FUNCTION_BLOCK FB_ST_HMICommand_Test EXTENDS TcUnit.FB_TestSuite
VAR_INPUT
END_VAR
VAR_OUTPUT
END_VAR
VAR
	testCommand : ST_HMICommand;
END_VAR

// Test runner - call all test methods
Test_InitialState();
Test_EnableCommand();
Test_DisableCommand();
Test_ResetCommand();
Test_StopCommand();
Test_TriggerCommand();
Test_ErrorCode();
Test_MultipleCommands();
Test_ClearCommands();

METHOD Test_ClearCommands
VAR_INPUT
END_VAR
TEST('Test_ClearCommands');

// Set all commands
testCommand.Enable := TRUE;
testCommand.Disable := TRUE;
testCommand.Reset := TRUE;
testCommand.Stop := TRUE;
testCommand.Trigger := TRUE;
testCommand.Error := 42;

// Clear all commands
testCommand.Enable := FALSE;
testCommand.Disable := FALSE;
testCommand.Reset := FALSE;
testCommand.Stop := FALSE;
testCommand.Trigger := FALSE;
testCommand.Error := 0;

// Verify all are cleared
AssertFalse(testCommand.Enable, 'Enable should be FALSE');
AssertFalse(testCommand.Disable, 'Disable should be FALSE');
AssertFalse(testCommand.Reset, 'Reset should be FALSE');
AssertFalse(testCommand.Stop, 'Stop should be FALSE');
AssertFalse(testCommand.Trigger, 'Trigger should be FALSE');
AssertEquals_BYTE(0, testCommand.Error, 'Error should be 0');

TEST_FINISHED();
END_METHOD

METHOD Test_DisableCommand
VAR_INPUT
END_VAR
TEST('Test_DisableCommand');

// Test Disable command can be set
testCommand.Disable := TRUE;
AssertTrue(testCommand.Disable, 'Disable should be TRUE when set');

// Reset
testCommand.Disable := FALSE;
AssertFalse(testCommand.Disable, 'Disable should be FALSE when reset');

TEST_FINISHED();
END_METHOD

METHOD Test_EnableCommand
VAR_INPUT
END_VAR
TEST('Test_EnableCommand');

// Test Enable command can be set
testCommand.Enable := TRUE;
AssertTrue(testCommand.Enable, 'Enable should be TRUE when set');

// Reset
testCommand.Enable := FALSE;
AssertFalse(testCommand.Enable, 'Enable should be FALSE when reset');

TEST_FINISHED();
END_METHOD

METHOD Test_ErrorCode
VAR_INPUT
END_VAR
TEST('Test_ErrorCode');

// Test Error code can be set to various values
testCommand.Error := 0;
AssertEquals_BYTE(0, testCommand.Error, 'Error should be 0');

testCommand.Error := 1;
AssertEquals_BYTE(1, testCommand.Error, 'Error should be 1');

testCommand.Error := 255;
AssertEquals_BYTE(255, testCommand.Error, 'Error should be 255');

testCommand.Error := 128;
AssertEquals_BYTE(128, testCommand.Error, 'Error should be 128');

TEST_FINISHED();
END_METHOD

METHOD Test_InitialState
VAR_INPUT
END_VAR
TEST('Test_InitialState');

// Test that all command flags are initially FALSE
testCommand.Enable := FALSE;
testCommand.Disable := FALSE;
testCommand.Reset := FALSE;
testCommand.Stop := FALSE;
testCommand.Trigger := FALSE;
testCommand.Error := 0;

AssertFalse(testCommand.Enable, 'Enable should be FALSE initially');
AssertFalse(testCommand.Disable, 'Disable should be FALSE initially');
AssertFalse(testCommand.Reset, 'Reset should be FALSE initially');
AssertFalse(testCommand.Stop, 'Stop should be FALSE initially');
AssertFalse(testCommand.Trigger, 'Trigger should be FALSE initially');
AssertEquals_BYTE(0, testCommand.Error, 'Error should be 0 initially');

TEST_FINISHED();
END_METHOD

METHOD Test_MultipleCommands
VAR_INPUT
END_VAR
TEST('Test_MultipleCommands');

// Test multiple commands can be set simultaneously
testCommand.Enable := TRUE;
testCommand.Trigger := TRUE;

AssertTrue(testCommand.Enable, 'Enable should be TRUE');
AssertTrue(testCommand.Trigger, 'Trigger should be TRUE');
AssertFalse(testCommand.Disable, 'Disable should remain FALSE');
AssertFalse(testCommand.Stop, 'Stop should remain FALSE');

TEST_FINISHED();
END_METHOD

METHOD Test_ResetCommand
VAR_INPUT
END_VAR
TEST('Test_ResetCommand');

// Test Reset command can be set
testCommand.Reset := TRUE;
AssertTrue(testCommand.Reset, 'Reset should be TRUE when set');

// Reset
testCommand.Reset := FALSE;
AssertFalse(testCommand.Reset, 'Reset should be FALSE when reset');

TEST_FINISHED();
END_METHOD

METHOD Test_StopCommand
VAR_INPUT
END_VAR
TEST('Test_StopCommand');

// Test Stop command can be set
testCommand.Stop := TRUE;
AssertTrue(testCommand.Stop, 'Stop should be TRUE when set');

// Reset
testCommand.Stop := FALSE;
AssertFalse(testCommand.Stop, 'Stop should be FALSE when reset');

TEST_FINISHED();
END_METHOD

METHOD Test_TriggerCommand
VAR_INPUT
END_VAR
TEST('Test_TriggerCommand');

// Test Trigger command can be set
testCommand.Trigger := TRUE;
AssertTrue(testCommand.Trigger, 'Trigger should be TRUE when set');

// Reset
testCommand.Trigger := FALSE;
AssertFalse(testCommand.Trigger, 'Trigger should be FALSE when reset');

TEST_FINISHED();
END_METHOD

END_FUNCTION_BLOCK

(* stored: Version 1.1.0.1
   POU FB_ST_HMICommand_Test: Id {a1111111-1111-1111-1111-111111111111}, SpecialFunc None
   Method Test_ClearCommands: Id {a1111111-1111-1111-1111-11111111111b}
   Method Test_DisableCommand: Id {a1111111-1111-1111-1111-111111111114}
   Method Test_EnableCommand: Id {a1111111-1111-1111-1111-111111111113}
   Method Test_ErrorCode: Id {a1111111-1111-1111-1111-111111111119}
   Method Test_InitialState: Id {a1111111-1111-1111-1111-111111111112}
   Method Test_MultipleCommands: Id {a1111111-1111-1111-1111-11111111111a}
   Method Test_ResetCommand: Id {a1111111-1111-1111-1111-111111111116}
   Method Test_StopCommand: Id {a1111111-1111-1111-1111-111111111117}
   Method Test_TriggerCommand: Id {a1111111-1111-1111-1111-111111111118} *)
